% RSLogix 500 project tripper_drbitboy.RSS, saved by version 8.30.00.16 %
PROJECT "UNTITLED"    % processor: Bul.1763 MicroLogix 1100 Series B %

PROGRAM FILES
  LAD 2   11 rungs

DATA FILES
  O0 OUTPUT  4 elements
  I1 INPUT  6 elements
  S2 STATUS  66 elements
  B3 BINARY  1 elements
  T4 TIMER  1 elements
  C5 COUNTER  1 elements
  R6 CONTROL  1 elements
  N7 INTEGER  1 elements
  F8 FLOAT  1 elements

LADDER 2
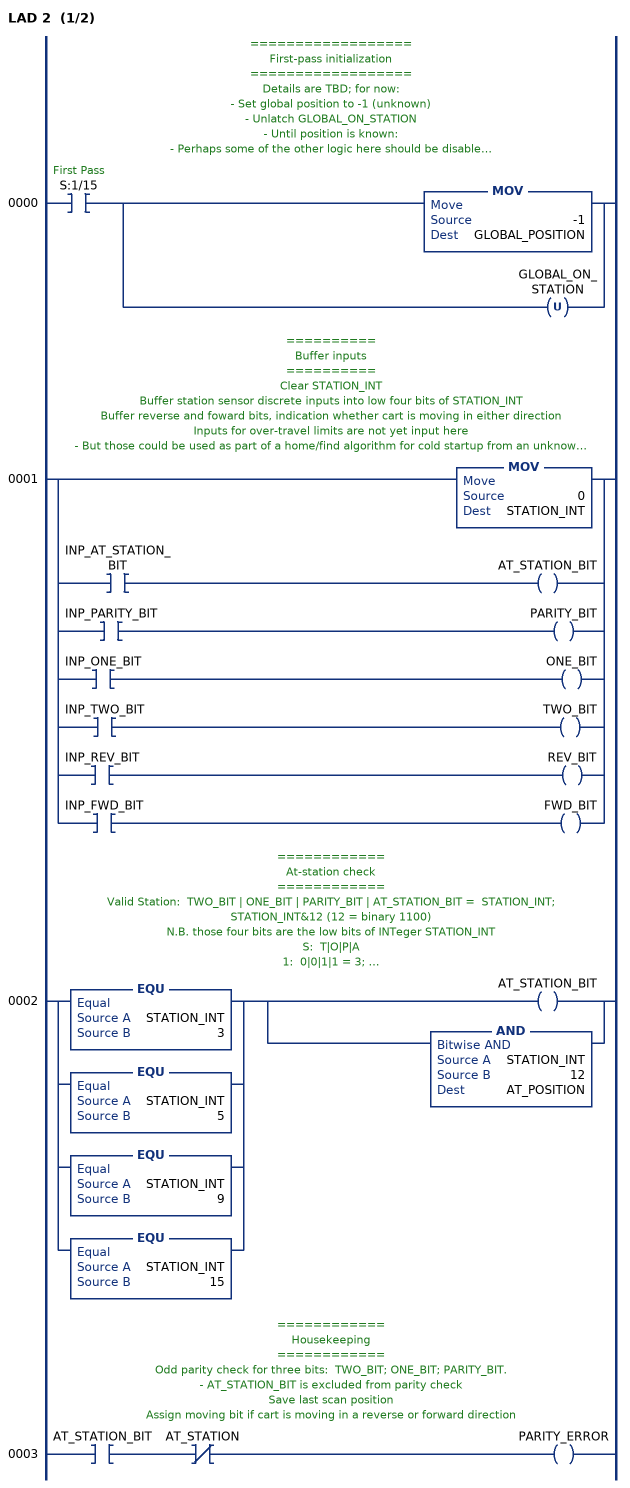
% Rung: 0 %  % edit flag set %
% ==================
% First-pass initialization
% ==================
% 
% Details are TBD; for now:
% - Set global position to -1 (unknown)
% - Unlatch GLOBAL_ON_STATION
% - Until position is known:
%   - Perhaps some of the other logic here should be disabled
%   - Perhaps only manual operation should be allowed, to find a position
%   - Perhaps a home action should be executed %
SOR XIC S:1/15 BST MOV -1 GLOBAL_POSITION NXB OTU GLOBAL_ON_STATION BND EOR
%   S:1/15  "First Pass" %
%   GLOBAL_POSITION   %
% Rung: 1 %  % edit flag set %
% ==========
% Buffer inputs
% ==========
% 
% Clear STATION_INT
% Buffer station sensor discrete inputs into low four bits of STATION_INT
% Buffer reverse and foward bits, indication whether cart is moving in either direction
% Inputs for over-travel limits are not yet input here
% - But those could be used as part of a home/find algorithm for cold startup from an unknown state %
SOR BST MOV 0 STATION_INT NXB XIC INP_AT_STATION_BIT OTE AT_STATION_BIT NXB XIC INP_PARITY_BIT OTE PARITY_BIT NXB XIC INP_ONE_BIT OTE ONE_BIT NXB XIC INP_TWO_BIT OTE TWO_BIT NXB XIC INP_REV_BIT OTE REV_BIT NXB XIC INP_FWD_BIT OTE FWD_BIT BND EOR
%   STATION_INT   %
%   INP_AT_STATION_BIT   %
%   AT_STATION_BIT   %
%   TWO_BIT   %
%   REV_BIT   %
%   INP_FWD_BIT   %
%   FWD_BIT   %
% Rung: 2 %  % edit flag set %
% ============
% At-station check
% ============
% 
% Valid Station:  TWO_BIT | ONE_BIT | PARITY_BIT | AT_STATION_BIT =  STATION_INT; STATION_INT&12 (12 = binary 1100)
% 
% N.B. those four bits are the low bits of INTeger STATION_INT
% 
% S:  T|O|P|A
% 1:  0|0|1|1 = 3; 0
% 2:  0|1|0|1 = 5; 4
% 3:  1|0|0|1 = 9; 8
% 4:  1|1|1|1 = 15; 12 %
SOR BST EQU STATION_INT 3 NXB EQU STATION_INT 5 NXB EQU STATION_INT 9 NXB EQU STATION_INT 15 BND BST OTE AT_STATION_BIT NXB AND STATION_INT 12 AT_POSITION BND EOR
%   STATION_INT   %
%   AT_STATION_BIT   %
% Rung: 3 %  % edit flag set %
% ============
% Housekeeping
% ============
% 
% Odd parity check for three bits:  TWO_BIT; ONE_BIT; PARITY_BIT.
% - AT_STATION_BIT is excluded from parity check
% Save last scan position
% Assign moving bit if cart is moving in a reverse or forward direction %
SOR XIC AT_STATION_BIT XIO AT_STATION OTE PARITY_ERROR EOR
%   AT_STATION_BIT   %
%   AT_STATION   %
%   PARITY_ERROR   %

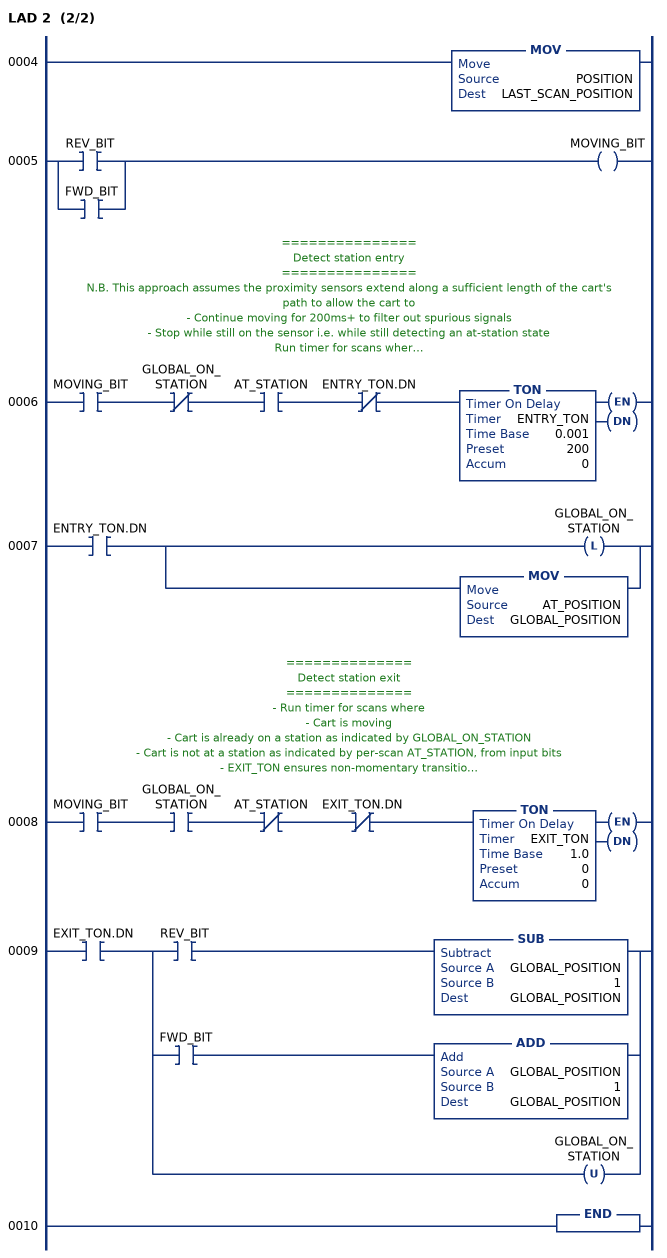
% Rung: 4 %  % edit flag set %
SOR MOV POSITION LAST_SCAN_POSITION EOR
%   POSITION   %
%   LAST_SCAN_POSITION   %
% Rung: 5 %  % edit flag set %
SOR BST XIC REV_BIT NXB XIC FWD_BIT BND OTE MOVING_BIT EOR
%   REV_BIT   %
%   FWD_BIT   %
%   MOVING_BIT   %
% Rung: 6 %  % edit flag set %
% ===============
% Detect station entry
% ===============
% 
% N.B. This approach assumes the proximity sensors extend along a sufficient length of the cart's path to allow the cart to
% - Continue moving for 200ms+ to filter out spurious signals
% - Stop while still on the sensor i.e. while still detecting an at-station state
% 
% Run timer for scans where
% - Cart is moving
% - Cart is not already on a station as indicated by GLOBAL_ON_STATION
% - Cart is at a station as indicated by per-scan AT_STATION, from input bits
% ENTRY_TON ensures non-momentary transition
% Entering a station is detected as expiry of ENTRY_TON
% - ENTRY_TON.DN will be a one-shot i.e. on for one scan
% - Assign global position
% - Latch GLOBAL_ON_STATION %
SOR XIC MOVING_BIT XIO GLOBAL_ON_STATION XIC AT_STATION XIO ENTRY_TON.DN TON ENTRY_TON 0.001 200 0 EOR
%   MOVING_BIT   %
%   AT_STATION   %
%   ENTRY_TON   %
% Rung: 7 %  % edit flag set %
SOR XIC ENTRY_TON.DN BST OTL GLOBAL_ON_STATION NXB MOV AT_POSITION GLOBAL_POSITION BND EOR
%   GLOBAL_POSITION   %
% Rung: 8 %  % edit flag set %
% ==============
% Detect station exit
% ==============
% 
% - Run timer for scans where
%   - Cart is moving
%   - Cart is already on a station as indicated by GLOBAL_ON_STATION
%   - Cart is not at a station as indicated by per-scan AT_STATION, from input bits
% - EXIT_TON ensures non-momentary transition
% - Exiting a station is detected as expiry of EXIT_TON
%   - EXIT_TON.DN will be a one-shot
%   - Decrement or increment global position
%   - Unlatch GLOBAL_ON_STATION %
SOR XIC MOVING_BIT XIC GLOBAL_ON_STATION XIO AT_STATION XIO EXIT_TON.DN TON EXIT_TON 1.0 0 0 EOR
%   MOVING_BIT   %
%   AT_STATION   %
% Rung: 9 %  % edit flag set %
SOR XIC EXIT_TON.DN BST XIC REV_BIT SUB GLOBAL_POSITION 1 GLOBAL_POSITION NXB XIC FWD_BIT ADD GLOBAL_POSITION 1 GLOBAL_POSITION NXB OTU GLOBAL_ON_STATION BND EOR
%   REV_BIT   %
%   GLOBAL_POSITION   %
%   FWD_BIT   %
% Rung: 10 %
SOR END EOR

OTHER DOCUMENTED ADDRESSES
  AT_TWO_BIT  
  OLD_POSITION  
  ON_STATION  
